// TIA Portal V18 export
FUNCTION_BLOCK "AlarmHandling"   // FB24, SCL
TITLE = Alarm handling
{ S7_Optimized_Access := 'TRUE' }
VERSION : 0.1
// Automatically generated alarm handling
// stored: AutoNumber true, IsIECCheckEnabled false, IsRetainMemResEnabled false, MemoryReserve 100, SetENOAutomatically false, UDAEnableTagReadback false
BEGIN
END_FUNCTION_BLOCK
